(*udt (user defined type) of Beckhoff EP9224 IP67 Block - Power Distribution Block, device commands
	To work in conjunction of udt_EP9224_CMDyymmdd
	auth. Brent Lekx-Toniolo of Sodecia GTAC; 

------------------------------------------------------------------------
REVISION NOTES:
	Version 20161207
		- Initial Concept
------------------------------------------------------------------------

*)


TYPE udt_EP9224_DEV_CMD_20161207 :
STRUCT

	Enable_Control_Via_Fieldbus: BOOL;
	Global_Reset: BOOL;

END_STRUCT
END_TYPE

(* stored: Version 1.1.0.1, ProductVersion 3.1.4024.9
   DUT udt_EP9224_DEV_CMD_20161207: Id {7d4218a8-2da1-4ea0-ade7-54abbf8c09e4} *)
